FUNCTION_BLOCK FB_MeinFunktionsbaustein
VAR_INPUT
	iMeinSensor1 AT %I* : BOOL;
	iMeinSensor2 AT %I* : BOOL;
 
END_VAR

iMeinSensor1 := TRUE;
iMeinSensor2 := TRUE;

END_FUNCTION_BLOCK

(* stored: Version 1.1.0.1, ProductVersion 3.1.4026.18
   POU FB_MeinFunktionsbaustein: Id {c8d2585c-13a7-4eee-8106-430e4a054763}, SpecialFunc None *)
